// TIA Portal project "009-sps-bandsteuerung-fb-ob-diagnose-tia-portal" (V17)

(* hardware
DEVICE "S7-300/ET200M-Station_1"  S7-300 station
   slot 0: "Profilschiene_0"  Rail  6ES7 390-1***0-0AA0
   slot 1: "PS 307 5A_1"  PS 307 5A  6ES7 307-1EA01-0AA0
   slot 2: "PLC_1"  CPU 314C-2 DP  6ES7 314-6CH04-0AB0  V3.3
      slot 0: "MPI-Schnittstelle_1"  MPI
      slot 1: "DP-Schnittstelle_1"  DP
      slot 2: "DI 24/DO 16_1"  DI24/DO16
      slot 3: "AI 5/AO 2_1"  AI5/AO2
      slot 4: "Zählen_1"  Counter
      slot 5: "Positionieren_1"  Positioning
   slot 4: "DI 16/DO 16x24VDC/0.5A_1"  DI16/DO16 x 24V / 0.5A  6ES7 323-1BL00-0AA0
   slot 5: "DI 16x24VDC_1"  DI16 x 24VDC  6ES7 321-1BH02-0AA0
   slot 6: "CP 342-5_1"  CP 342-5  6GK7 342-5DA03-0XE0  V6.0
   slot 7: "CP 343-1_1"  CP 343-1  6GK7 343-1EX30-0XE0  V2.0
*)

// ===== PLC "PLC_1"  CPU 314C-2 DP =====

VAR_GLOBAL   // PLC tag table "Standard-Variablentabelle"
   "Tag_3" AT %M255.1 : Bool;
   "Start" AT %E0.0 : Bool;
   "Tag_4" AT %M0.0 : Bool;
   "Tag_5" AT %MD10 : DWord;
   "Tag_6" AT %M20.0 : Bool;
   "Tag_7" AT %M0.1 : Bool;
   "Tag_8" AT %M0.2 : Bool;
   "Tag_1" AT %MD30 : DWord;
   "Ausgang" AT %AW0 : Word;
   "Tag_2" AT %AW2 : Word;
   "Tag_9" AT %M255.5 : Bool;
   "Tag_10" AT %M255.3 : Bool;
   "Tag_11" AT %A0.0 : Bool;
   "Tag_12" AT %A124.0 : Bool;
   "Tag_13" AT %A125.0 : Bool;
   "Tag_14" AT %A0.1 : Bool;
END_VAR

DATA_BLOCK "FB10 Bandsteuerung_DB"   // DB1
{ S7_Optimized_Access := 'FALSE' }
VERSION : 0.1
// stored: InstanceOfName FB10 Bandsteuerung
"FB10 Bandsteuerung"
BEGIN
END_DATA_BLOCK

DATA_BLOCK "xdb100 VAR"   // DB100
{ S7_Optimized_Access := 'FALSE' }
VERSION : 0.1
   VAR
      "s_OB100 ok" : String[10] := 'OB 100 OK';
      s_Message : String[10] := '';
      s_Clear : String[10] := '';
      x_clear : Bool;
      di_valOB10 : DInt;
      di_valOB32 : DInt;
      "OB20 ok" : String[10] := 'OB20 OK';
      Mekdung : String[10];
      x_startSFC32 : Bool;
      s_OB121OK : String[10] := 'OB121 OK';
   END_VAR
BEGIN
END_DATA_BLOCK

DATA_BLOCK "xdb100 VAR_1"   // DB101
{ S7_Optimized_Access := 'FALSE' }
VERSION : 0.1
   VAR
      "s_OB100 ok" : String[10] := 'OB 100 OK';
      s_Message : String[10] := '';
      s_Clear : String[10] := '';
      x_clear : Bool;
      di_valOB10 : DInt;
      di_valOB32 : DInt;
      "OB20 ok" : String[10] := 'OB20 OK';
      Mekdung : String[10];
      x_startSFC32 : Bool;
      dummy : Bool;
      dummy_1 : Bool;
   END_VAR
BEGIN
END_DATA_BLOCK

FUNCTION_BLOCK "FB10 Bandsteuerung"   // FB10, FBD
{ S7_Optimized_Access := 'FALSE' }
VERSION : 0.1
   VAR_INPUT
      x_MainSwitch_S1 : Bool;
      x_Mod_Switch : Bool;
      x_Break : Bool;
      x_Direction : Bool;
      x_v1 : Bool;
      x_v2 : Bool;
      x_v3 : Bool;
      x_EMO : Bool;
      x_Reset : Bool;
      clock : Bool;
   END_VAR
   VAR_OUTPUT
      x_Main_Switch_Ctrl : Bool;
      x_Mod_Switch_Ctrl : Bool;
      x_Break_Ctrl : Bool;
      x_Dir_Ctrl : Bool;
      x_v1_Ctrl : Bool;
      x_v2_Ctrl : Bool;
      x_v3_Ctrl : Bool;
      x_EMO_Ctrl : Bool;
      x_Reset_Ctrl : Bool;
      x_Motor_On : Bool;
      x_Mot_Left : Bool;
      x_Mot_Break_off : Bool;
      x_Velo_3 : Bool;
      x_Velo_2 : Bool;
      x_Velo_1 : Bool;
      "x_Mod A/D" : Bool;
      x_R_LED3 : Bool;
      x_R_LED2 : Bool;
      x_R_LED1 : Bool;
      x_Mot_Akt_LED : Bool;
      x_L_LED1 : Bool;
      x_L_LED2 : Bool;
      x_L_LED3 : Bool;
      w_Clear_w0 : Word;
      w_Clear_w124 : Word;
   END_VAR
   VAR
      x_EMO_SR : Bool;
      x_ptrig_EMO : Bool;
      x_dummy : Bool;
   END_VAR
   VAR_TEMP   // added for the SCL form of the ladder/FBD networks
      _w1 : Bool;
   END_VAR
BEGIN

REGION Network 1: Emo
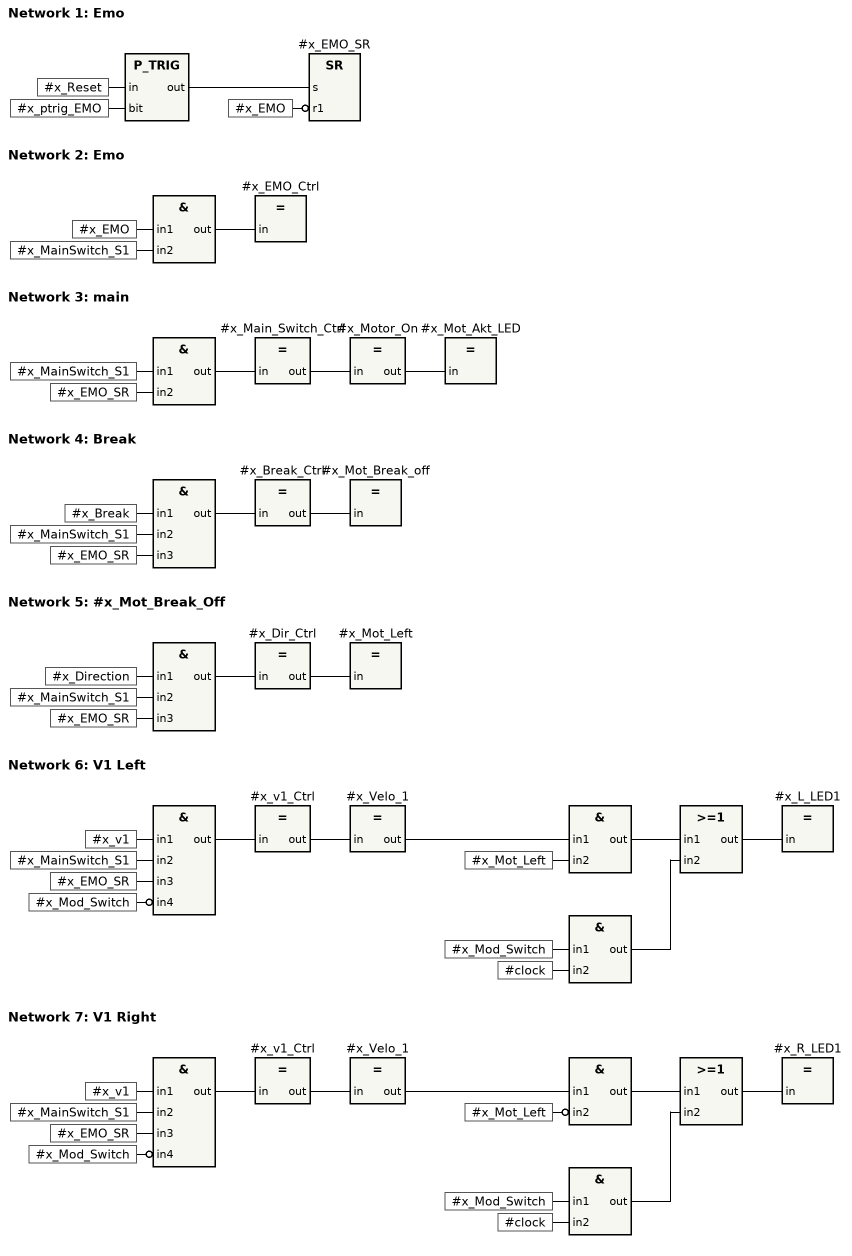
   #_w1 := #x_Reset AND NOT #x_ptrig_EMO;   // rising edge
   #x_ptrig_EMO := #x_Reset;
   IF #_w1 THEN
       #x_EMO_SR := TRUE;   // SR flip-flop
   END_IF;
   IF NOT #x_EMO THEN #x_EMO_SR := FALSE; END_IF;
END_REGION

REGION Network 2: Emo
   #x_EMO_Ctrl := #x_EMO AND #x_MainSwitch_S1;
END_REGION

REGION Network 3: main
   #x_Main_Switch_Ctrl := #x_MainSwitch_S1 AND #x_EMO_SR;
   #x_Motor_On := #x_Main_Switch_Ctrl;
   #x_Mot_Akt_LED := #x_Main_Switch_Ctrl;
END_REGION

REGION Network 4: Break
   #x_Break_Ctrl := #x_Break AND #x_MainSwitch_S1 AND #x_EMO_SR;
   #x_Mot_Break_off := #x_Break_Ctrl;
END_REGION

REGION Network 5: #x_Mot_Break_Off
   #x_Dir_Ctrl := #x_Direction AND #x_MainSwitch_S1 AND #x_EMO_SR;
   #x_Mot_Left := #x_Dir_Ctrl;
END_REGION

REGION Network 6: V1 Left
   #x_v1_Ctrl := #x_v1 AND #x_MainSwitch_S1 AND #x_EMO_SR AND NOT #x_Mod_Switch;
   #x_Velo_1 := #x_v1_Ctrl;
   #x_L_LED1 := (#x_v1_Ctrl AND #x_Mot_Left) OR (#x_Mod_Switch AND #clock);
END_REGION

REGION Network 7: V1 Right
   #x_v1_Ctrl := #x_v1 AND #x_MainSwitch_S1 AND #x_EMO_SR AND NOT #x_Mod_Switch;
   #x_Velo_1 := #x_v1_Ctrl;
   #x_R_LED1 := (#x_v1_Ctrl AND NOT #x_Mot_Left) OR (#x_Mod_Switch AND #clock);
END_REGION

REGION Network 8: V2 Left
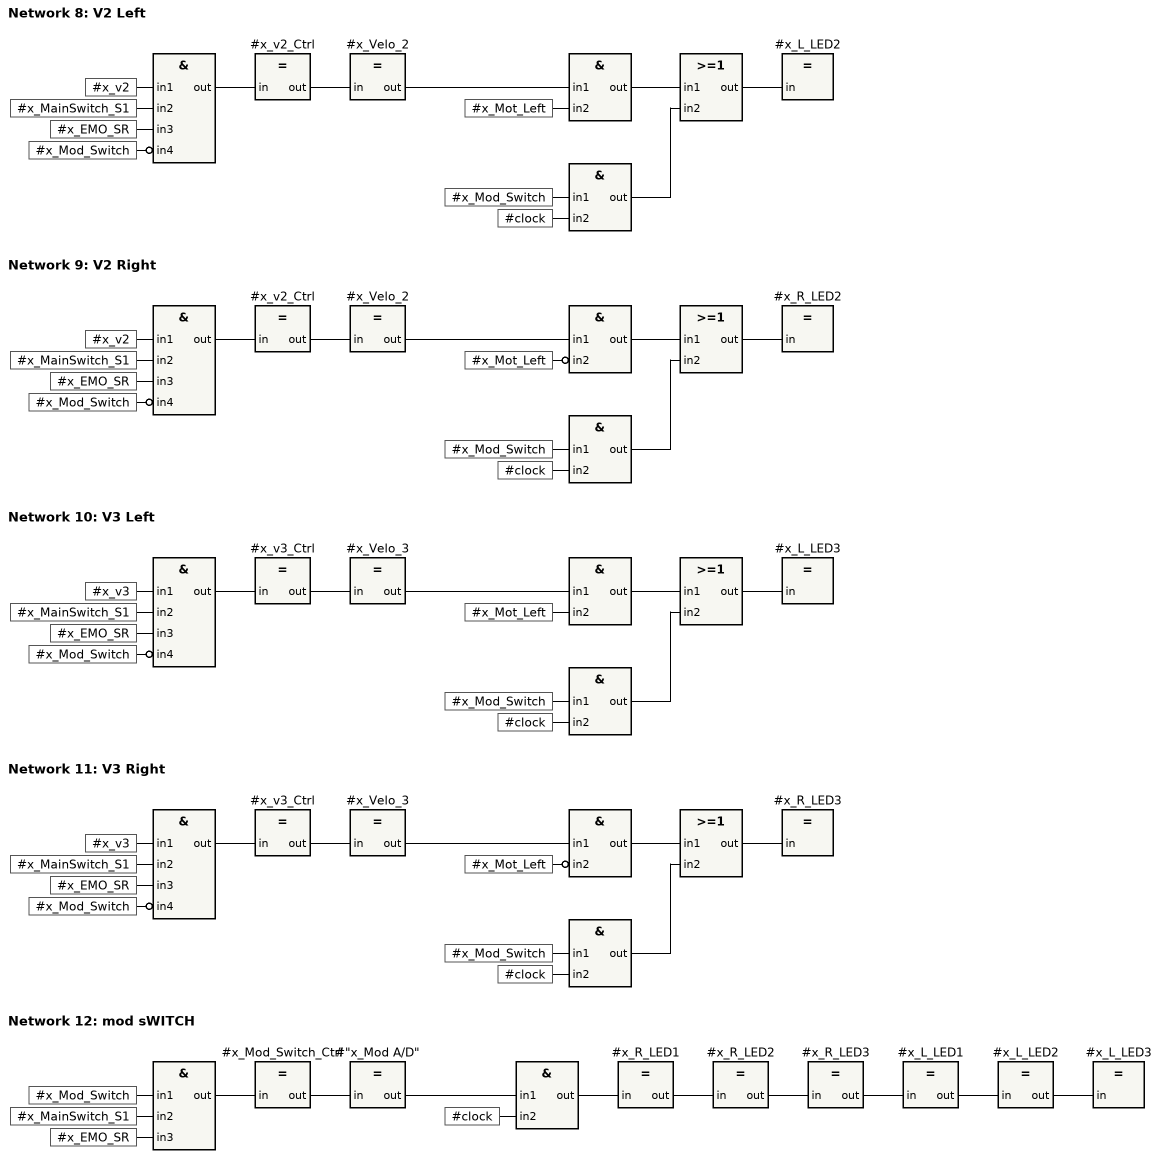
   #x_v2_Ctrl := #x_v2 AND #x_MainSwitch_S1 AND #x_EMO_SR AND NOT #x_Mod_Switch;
   #x_Velo_2 := #x_v2_Ctrl;
   #x_L_LED2 := (#x_v2_Ctrl AND #x_Mot_Left) OR (#x_Mod_Switch AND #clock);
END_REGION

REGION Network 9: V2 Right
   #x_v2_Ctrl := #x_v2 AND #x_MainSwitch_S1 AND #x_EMO_SR AND NOT #x_Mod_Switch;
   #x_Velo_2 := #x_v2_Ctrl;
   #x_R_LED2 := (#x_v2_Ctrl AND NOT #x_Mot_Left) OR (#x_Mod_Switch AND #clock);
END_REGION

REGION Network 10: V3 Left
   #x_v3_Ctrl := #x_v3 AND #x_MainSwitch_S1 AND #x_EMO_SR AND NOT #x_Mod_Switch;
   #x_Velo_3 := #x_v3_Ctrl;
   #x_L_LED3 := (#x_v3_Ctrl AND #x_Mot_Left) OR (#x_Mod_Switch AND #clock);
END_REGION

REGION Network 11: V3 Right
   #x_v3_Ctrl := #x_v3 AND #x_MainSwitch_S1 AND #x_EMO_SR AND NOT #x_Mod_Switch;
   #x_Velo_3 := #x_v3_Ctrl;
   #x_R_LED3 := (#x_v3_Ctrl AND NOT #x_Mot_Left) OR (#x_Mod_Switch AND #clock);
END_REGION

REGION Network 12: mod sWITCH
   #x_Mod_Switch_Ctrl := #x_Mod_Switch AND #x_MainSwitch_S1 AND #x_EMO_SR;
   #"x_Mod A/D" := #x_Mod_Switch_Ctrl;
   #x_R_LED1 := #x_Mod_Switch_Ctrl AND #clock;
   #x_R_LED2 := #x_R_LED1;
   #x_R_LED3 := #x_R_LED1;
   #x_L_LED1 := #x_R_LED1;
   #x_L_LED2 := #x_R_LED1;
   #x_L_LED3 := #x_R_LED1;
END_REGION
END_FUNCTION_BLOCK

ORGANIZATION_BLOCK "Main"   // OB1, FBD
TITLE = "Main Program Sweep (Cycle)"
{ S7_Optimized_Access := 'FALSE' }
VERSION : 0.1
   VAR_TEMP
      OB1_EV_CLASS : Byte;   // Bits 0-3 = 1 (Coming event), Bits 4-7 = 1 (Event class 1)
      OB1_SCAN_1 : Byte;   // 1 (Cold restart scan 1 of OB 1), 3 (Scan 2-n of OB 1)
      OB1_PRIORITY : Byte;   // Priority of OB Execution
      OB1_OB_NUMBR : Byte;   // 1 (Organization block 1, OB1)
      OB1_RESERVED_1 : Byte;   // Reserved for system
      OB1_RESERVED_2 : Byte;   // Reserved for system
      OB1_PREV_CYCLE : Int;   // Cycle time of previous OB1 scan (milliseconds)
      OB1_MIN_CYCLE : Int;   // Minimum cycle time of OB1 (milliseconds)
      OB1_MAX_CYCLE : Int;   // Maximum cycle time of OB1 (milliseconds)
      OB1_DATE_TIME : Date_And_Time;   // Date and time OB1 started
      ret : Int;
   END_VAR
BEGIN

REGION Network 1
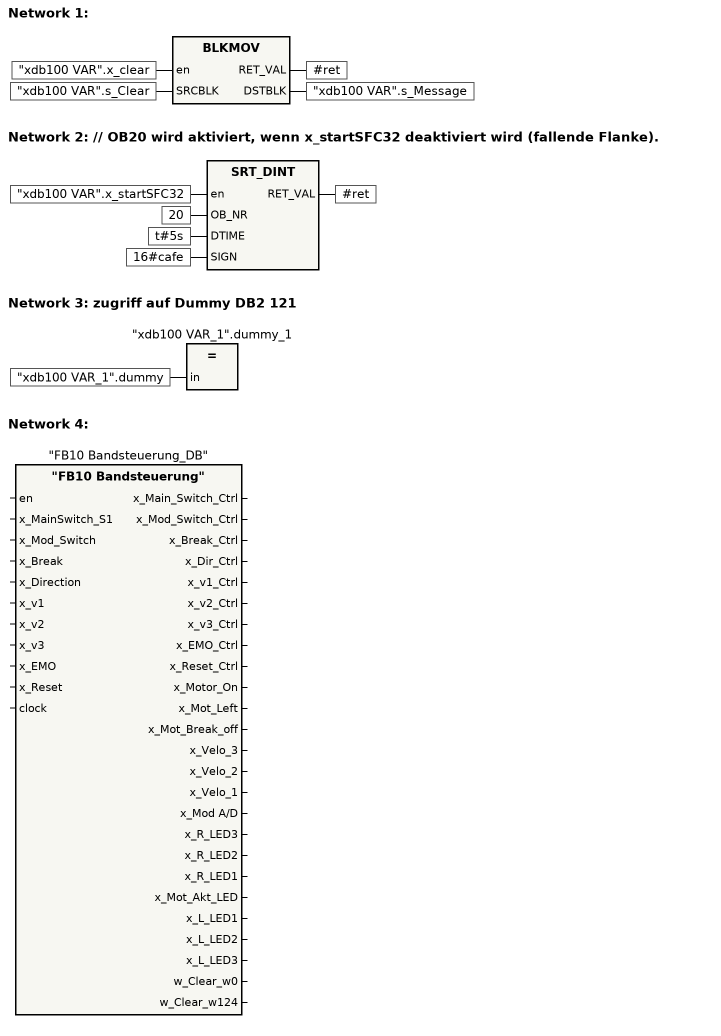
   IF "xdb100 VAR".x_clear THEN
       #ret := BLKMOV(SRCBLK := "xdb100 VAR".s_Clear, DSTBLK => "xdb100 VAR".s_Message);
   END_IF;
END_REGION

REGION Network 2: // OB20 wird aktiviert, wenn x_startSFC32 deaktiviert wird (fallende Flanke).
   IF "xdb100 VAR".x_startSFC32 THEN #ret := SRT_DINT(OB_NR := 20, DTIME := t#5s, SIGN := 16#cafe); END_IF;
END_REGION

REGION Network 3: zugriff auf Dummy DB2 121
   // // Zugriff auf den Dummy-DB101 (Wenn fehler passiert)
   // zbs:
   // // Wird DB101 während des RUN-Betriebs gelöscht, wird OB121 aufgrund eines Programmierfehlers aufgerufen.
   "xdb100 VAR_1".dummy_1 := "xdb100 VAR_1".dummy;
END_REGION

REGION Network 4
   "FB10 Bandsteuerung_DB"();   // "FB10 Bandsteuerung"
END_REGION
END_ORGANIZATION_BLOCK

ORGANIZATION_BLOCK "TOD_INTO"   // OB10, FBD
TITLE = "Time of Day Interrupt"
{ S7_Optimized_Access := 'FALSE' }
VERSION : 0.1
   VAR_TEMP
      OB10_EV_CLASS : Byte;   // Bits 0-3 = 1 (Coming event), Bits 4-7 = 1 (Event class 1)
      OB10_STRT_INFO : Byte;   // 16#11 (OB 10 has started)
      OB10_PRIORITY : Byte;   // Priority of OB Execution
      OB10_OB_NUMBR : Byte;   // 10 (Organization block 10, OB10)
      OB10_RESERVED_1 : Byte;   // Reserved for system
      OB10_RESERVED_2 : Byte;   // Reserved for system
      OB10_PERIOD_EXE : Word;   // Period of execution (once, per minute/hour/day/week/month/year)
      OB10_RESERVED_3 : Int;   // Reserved for system
      OB10_RESERVED_4 : Int;   // Reserved for system
      OB10_DATE_TIME : Date_And_Time;   // Date and time OB10 started
   END_VAR
BEGIN

REGION Network 1
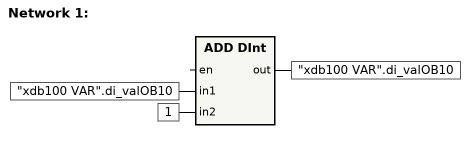
   "xdb100 VAR".di_valOB10 := "xdb100 VAR".di_valOB10 + 1;
END_REGION
END_ORGANIZATION_BLOCK

ORGANIZATION_BLOCK "Verzörungsalarm"   // OB20, FBD
TITLE = "Time Delay Interrupt"
{ S7_Optimized_Access := 'FALSE' }
VERSION : 0.1
   VAR_TEMP
      OB20_EV_CLASS : Byte;   // Bits 0-3 = 1 (Coming event), Bits 4-7 = 1 (Event class 1)
      OB20_STRT_INF : Byte;   // 16#21 (OB 20 has started)
      OB20_PRIORITY : Byte;   // Priority of OB Execution
      OB20_OB_NUMBR : Byte;   // 20 (Organization block 20, OB20)
      OB20_RESERVED_1 : Byte;   // Reserved for system
      OB20_RESERVED_2 : Byte;   // Reserved for system
      OB20_SIGN : Word;   // Identifier input (SIGN) attached to SRT_DINT
      OB20_DTIME : Time;   // Delay time (DTIME) input to SRT_DINT instruction
      OB20_DATE_TIME : Date_And_Time;   // Date and time OB20 started
      ret : Int;
   END_VAR
BEGIN

REGION Network 1
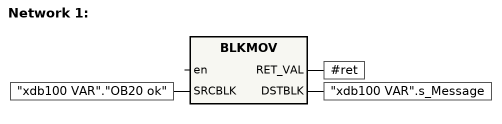
   #ret := BLKMOV(SRCBLK := "xdb100 VAR"."OB20 ok", DSTBLK => "xdb100 VAR".s_Message);
END_REGION
END_ORGANIZATION_BLOCK

ORGANIZATION_BLOCK "Weckalarm1000ms"   // OB32, FBD
TITLE = "Cyclic Interrupt"
{ S7_Optimized_Access := 'FALSE' }
VERSION : 0.1
   VAR_TEMP
      OB32_EV_CLASS : Byte;   // Bits 0-3 = 1 (Coming event), Bits 4-7 = 1 (Event class 1)
      OB32_STRT_INF : Byte;   // 16#33 (OB 32 has started)
      OB32_PRIORITY : Byte;   // Priority of OB Execution
      OB32_OB_NUMBR : Byte;   // 32 (Organization block 32, OB32)
      OB32_RESERVED_1 : Byte;   // Reserved for system
      OB32_RESERVED_2 : Byte;   // Reserved for system
      OB32_PHS_OFFSET : Int;   // Phase offset (integer, milliseconds)
      OB32_RESERVED_3 : Int;   // Reserved for system
      OB32_EXC_FREQ : Int;   // Frequency of execution (msec)
      OB32_DATE_TIME : Date_And_Time;   // Date and time OB32 started
   END_VAR
BEGIN

REGION Network 1
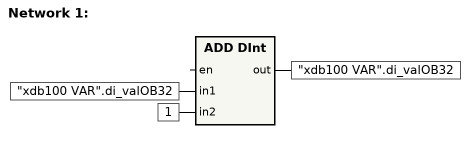
   "xdb100 VAR".di_valOB32 := "xdb100 VAR".di_valOB32 + 1;
END_REGION
END_ORGANIZATION_BLOCK

ORGANIZATION_BLOCK "COMPLETE RESTART"   // OB100, FBD
TITLE = "Complete Restart"
{ S7_Optimized_Access := 'FALSE' }
VERSION : 0.1
   VAR_TEMP
      OB100_EV_CLASS : Byte;   // 16#13, Event class 1, Entering event state, Event logged in diagnostic buffer
      OB100_STRTUP : Byte;   // 16#81/82/83/84 Method of startup
      OB100_PRIORITY : Byte;   // Priority of OB Execution
      OB100_OB_NUMBR : Byte;   // 100 (Organization block 100, OB100)
      OB100_RESERVED_1 : Byte;   // Reserved for system
      OB100_RESERVED_2 : Byte;   // Reserved for system
      OB100_STOP : Word;   // Event that caused CPU to stop (16#4xxx)
      OB100_STRT_INFO : DWord;   // Information on how system started
      OB100_DATE_TIME : Date_And_Time;   // Date and time OB100 started
      ret : Int;
   END_VAR
BEGIN

REGION Network 1
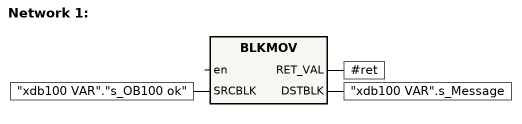
   #ret := BLKMOV(SRCBLK := "xdb100 VAR"."s_OB100 ok", DSTBLK => "xdb100 VAR".s_Message);
END_REGION
END_ORGANIZATION_BLOCK

ORGANIZATION_BLOCK "PROG_ERR"   // OB121, FBD
TITLE = "Programming Error"
{ S7_Optimized_Access := 'FALSE' }
VERSION : 0.1
   VAR_TEMP
      OB121_EV_CLASS : Byte;   // 16#25, Event class 2, Entering event state, Internal fault event
      OB121_SW_FLT : Byte;   // 16#XX Software programming fault
      OB121_PRIORITY : Byte;   // Priority of OB Execution
      OB121_OB_NUMBR : Byte;   // 121 (Organization block 121, OB121)
      OB121_BLK_TYPE : Byte;   // 16#88/8A/8B/8C/8E Type of block fault occured in
      OB121_RESERVED_1 : Byte;   // Reserved for system
      OB121_FLT_REG : Word;   // 16#XX Specific register that caused fault
      OB121_BLK_NUM : Word;   // Number of block that programming fault occured in
      OB121_PRG_ADDR : Word;   // Address in block where programming fault occured
      OB121_DATE_TIME : Date_And_Time;   // Date and time OB121 started
      ret : Int;
   END_VAR
BEGIN

REGION Network 1
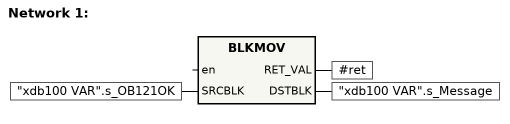
   #ret := BLKMOV(SRCBLK := "xdb100 VAR".s_OB121OK, DSTBLK => "xdb100 VAR".s_Message);
END_REGION
END_ORGANIZATION_BLOCK